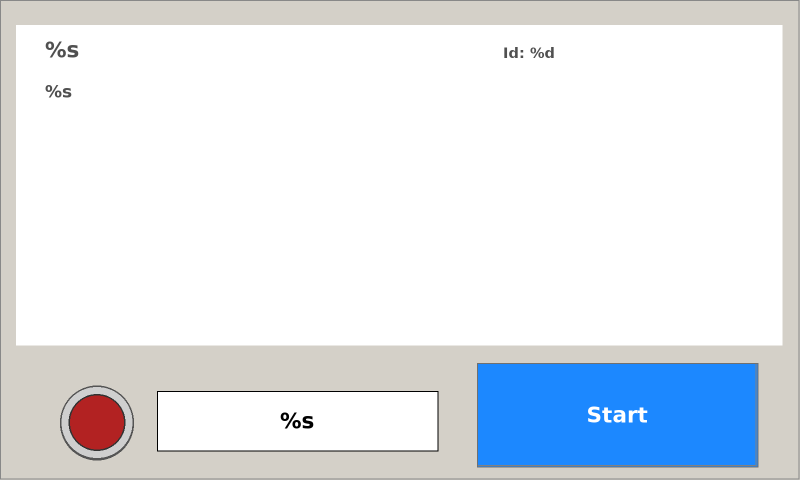
VISUALIZATION Tower1  // 800x480
    Button (110,230 150x110), "Down"
    Button (110,90 150x110), "Up"
    Button (110,90 150x110), "Up", invisible if: NOT(MAIN.Machine.Tower.Enabled)
        tap MAIN.Machine.Tower.backwardButton
    Button (110,230 150x110), "Down", invisible if: GVL.eMachineState = E_MachineState.Error OR NOT(MAIN.Machine.Tower.Enabled)
        tap MAIN.Machine.Tower.forwardButton
    Rectangle (608,99 110x50), "Low", invisible if: GVL.UI_EnableHighSpeed = False
        toggle GVL.UI_EnableHighSpeed
    Rectangle (608,99 110x50), "High", invisible if: GVL.eMachineState = E_MachineState.Error or GVL.UI_EnableHighSpeed = True
        toggle GVL.UI_EnableHighSpeed
    Label (2039,520 94x27), "Position", invisible if: GVL.eMachineState = E_MachineState.Error
    RoundedRectangle (2039,555 137x23), "%1.2f m", text variable: MAIN.Machine.Tower.ActualPos, invisible if: GVL.eMachineState = E_MachineState.Error
    Label (459,79 139x27), "Speed:"
    RoundedRectangle (460,109 96x36), "%s", text variable: TO_STRING(MAIN.Machine.Tower.SpeedSetting)
    Lamp1 (45,381 104x85), variable: MAIN.Machine.Tower.light_pulse, invisible if: GVL.eMachineState = E_MachineState.Error, style: Lamp-Lamp1-Green
    RoundedRectangle (157,391 281x60), "%s", text variable: TO_STRING(GVL.eMachineState)
    Button (477,363 281x104), "Stop", invisible if: GVL.eMachineState = E_MachineState.Error OR GVL.eMachineState = E_MachineState.Ready
        tap MAIN.Machine.Tower.stopButton
    Lamp1 (45,380 104x85), variable: MAIN.Machine.Tower.light_pulse, invisible if: NOT(GVL.eMachineState = E_MachineState.Error), style: Lamp-Lamp1-Red
    Button (477,363 281x104), "Reset", invisible if: NOT(GVL.eMachineState = E_MachineState.Error)
        tap MAIN.Machine.Tower.resetButton
    Button (477,363 281x104), "Start", invisible if: GVL.eMachineState = E_MachineState.Error OR MAIN.Machine.Tower.Enabled OR MAIN.Machine.Tower.Enabled
        tap MAIN.Machine.Tower.startButton
    Rectangle (16,25 766x320), invisible if: NOT(GVL.eMachineState = E_MachineState.Error)
    Rectangle (42,80 600x105), "%s", text variable: MAIN.Machine.Tower.mc_error_string, invisible if: NOT(GVL.eMachineState = E_MachineState.Error)
    Rectangle (42,27 452x46), "%s", text variable: MAIN.Machine.Tower.error_header_string, invisible if: NOT(GVL.eMachineState = E_MachineState.Error)
    Rectangle (500,30 136x46), "Id: %d", text variable: MAIN.Machine.Tower.mc_errorID, invisible if: NOT(GVL.eMachineState = E_MachineState.Error)
END_VISUALIZATION

(* stored: Version 1.1.0.1, ProductVersion 3.1.4024.9
   Visu Tower1: Id {6baabd85-cc70-46b4-b7be-18493bcb535e} *)
